{attribute 'linkalways'} 
{attribute 'no_explicit_call' := 'This FB is a CLASS and must be accessed using methods or properties'}
{attribute 'enable_dynamic_creation'}
FUNCTION_BLOCK JsonDomNavigator IMPLEMENTS I_JsonPathVisitor
VAR
	jsonDomParser : REFERENCE TO JsonDomParser;
	currentJsonPosition : SJsonValue;
	_currentNode : SJsonValue;
END_VAR

METHOD ArrayIndexFound
VAR_INPUT
	Index : UDINT;
END_VAR
currentJsonPosition := jsonDomParser.GetArrayValueByIdx(currentJsonPosition, Index);
END_METHOD

PROPERTY PUBLIC CurrentNode : SJsonValue
GET
CurrentNode := _currentNode;
END_GET
END_PROPERTY

METHOD EndOfParse
VAR_INPUT
END_VAR
_currentNode := currentJsonPosition;
END_METHOD

METHOD FB_init : BOOL
VAR_INPUT
	bInitRetains : BOOL; // if TRUE, the retain variables are initialized (warm start / cold start)
	bInCopyCode : BOOL;  // if TRUE, the instance afterwards gets moved into the copy code (online change)
	JsonDomParser : REFERENCE TO JsonDomParser;
END_VAR
THIS^.jsonDomParser REF= JsonDomParser;
END_METHOD

METHOD InvalidSyntaxFound
VAR_INPUT
	Character : BYTE;
	Position : UDINT;
END_VAR
currentJsonPosition := 0;
END_METHOD

METHOD PropertyFound
VAR_INPUT
	Name : T_MAXSTRING;
END_VAR
currentJsonPosition := jsonDomParser.FindMember(currentJsonPosition,Name);
END_METHOD

METHOD StartOfParse
VAR_INPUT
END_VAR
currentJsonPosition := jsonDomParser.GetDocumentRoot();
END_METHOD

END_FUNCTION_BLOCK

(* stored: Version 1.1.0.1, ProductVersion 3.1.4024.12
   POU JsonDomNavigator: Id {17a0dbe1-b117-4cf7-a87e-789019e1809b}, SpecialFunc None
   Folder Constructor: Id {9e9629ff-a170-4d6e-9893-343ba96c6ab5}
   Method ArrayIndexFound: Id {02b14946-dad5-475b-9a74-4887cebcfcf0}
   Property CurrentNode: Id {02f0a770-75f1-4caf-be18-1a778c9ef0a0}
   Get Get: Id {8afa67d9-7ddb-4a7e-9ee2-aea4c8e52d50}
   Method EndOfParse: Id {835925b2-376e-48d1-9ffc-3e685f01d04f}
   Method FB_init: Id {53b46c59-779c-41e8-b0f2-d9c79903517f}
   Method InvalidSyntaxFound: Id {9ac2fe37-8d3e-4f3f-b75c-762a5d41031f}
   Method PropertyFound: Id {9919dff6-0bc9-4fe7-9d9c-e6f157a227e6}
   Method StartOfParse: Id {b0226ba8-b6c8-4fd7-ada7-3f05f8bd9ad5} *)
